SUBAPPLICATION GetEndpointFromOrchestrationOpcUaFull (* Get the endpoint at INDEX from a request orchestration response *)
  (* Standard: 61499-2; Description: Copyright (c) 2019 fortiss GmbH This program and the accompanying materials are made available under the terms of the Eclipse Public License 2.0 which is available at https://www.eclipse.org/legal/epl-2.0/ SPDX-License-Identifier: EPL-2.0 *)
  (* Version 1.0, 2019-09-17, Jose Cabral, fortiss GmbH *)
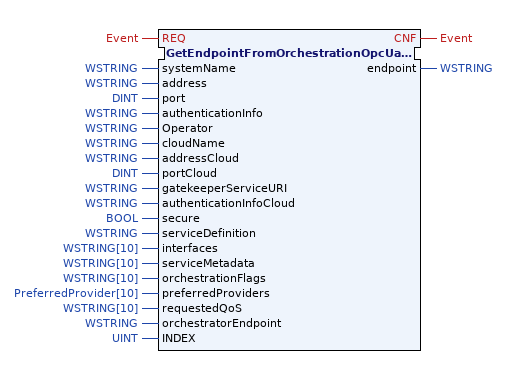
  EVENT_INPUT
    REQ; (* Request orchestration *)
  END_EVENT
  EVENT_OUTPUT
    CNF; (* Request finished *)
  END_EVENT
  VAR_INPUT
    systemName : WSTRING; (* Identification of the system *)
    address : WSTRING; (* Address of the offered services *)
    port : DINT; (* Port of the of the offered services *)
    authenticationInfo : WSTRING; (* Authentication info of the system *)
    Operator : WSTRING; (* Company (the capital  O is to avoid clash when exporting to C++) *)
    cloudName : WSTRING; (* Identification of the cloud *)
    addressCloud : WSTRING; (* Address to access the cloud *)
    portCloud : DINT; (* Port to access the cloud *)
    gatekeeperServiceURI : WSTRING; (* (Unclear documentation) *)
    authenticationInfoCloud : WSTRING; (* Authentication info of the cloud *)
    secure : BOOL; (* (Unclear documentation) *)
    serviceDefinition : WSTRING; (* Identification of the service *)
    interfaces : ARRAY [0..9] OF WSTRING; (* Interfaces implemented by the service *)
    serviceMetadata : ARRAY [0..9] OF WSTRING; (* Metadata of the service in key=value format *)
    orchestrationFlags : ARRAY [0..9] OF WSTRING; (* These flags can be set to tailor the orchestration process (use just the names of the flags to be enabled) *)
    preferredProviders : ARRAY [0..9] OF PreferredProvider; (* There can be a list from the Consumer stating which other Application Systems (even from other Clouds) it wishes to connect. If this field is filled out, the Orchestrator will try to facilitate these preferences *)
    requestedQoS : ARRAY [0..9] OF WSTRING; (* This object will be presenting the Consumer’s selected QoS level. Not implemented *)
    orchestratorEndpoint : WSTRING; (* Enpoint of the orchestrator *)
    INDEX : UINT; (* Position in the array of the requested forms *)
  END_VAR
  VAR_OUTPUT
    endpoint : WSTRING; (* Endpoint at position INDEX from orchestration forms *)
  END_VAR
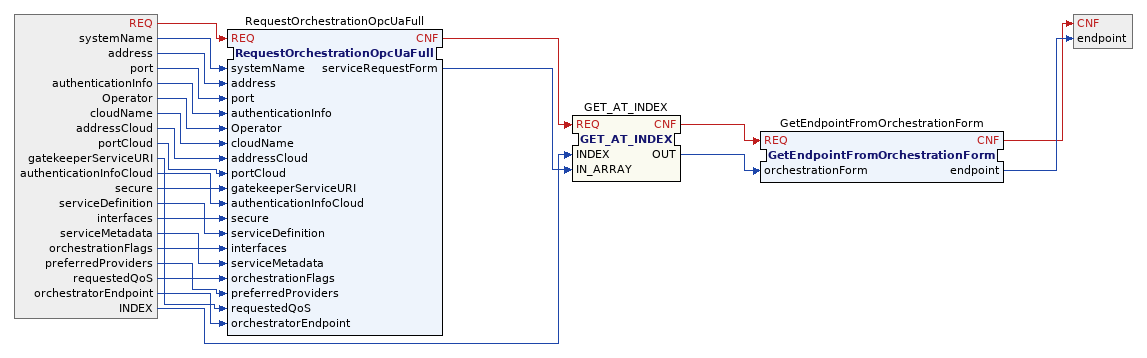
  FBS
    GET_AT_INDEX : GET_AT_INDEX;
  END_FBS
  SUBAPPS
    GetEndpointFromOrchestrationForm : GetEndpointFromOrchestrationForm;
    RequestOrchestrationOpcUaFull : RequestOrchestrationOpcUaFull;
  END_SUBAPPS
  EVENT_CONNECTIONS
    GET_AT_INDEX.CNF TO GetEndpointFromOrchestrationForm.REQ;
    GetEndpointFromOrchestrationForm.CNF TO CNF;
    REQ TO RequestOrchestrationOpcUaFull.REQ;
    RequestOrchestrationOpcUaFull.CNF TO GET_AT_INDEX.REQ;
  END_CONNECTIONS
  DATA_CONNECTIONS
    GET_AT_INDEX.OUT TO GetEndpointFromOrchestrationForm.orchestrationForm;
    INDEX TO GET_AT_INDEX.INDEX;
    GetEndpointFromOrchestrationForm.endpoint TO endpoint;
    systemName TO RequestOrchestrationOpcUaFull.systemName;
    address TO RequestOrchestrationOpcUaFull.address;
    port TO RequestOrchestrationOpcUaFull.port;
    authenticationInfo TO RequestOrchestrationOpcUaFull.authenticationInfo;
    Operator TO RequestOrchestrationOpcUaFull.Operator;
    cloudName TO RequestOrchestrationOpcUaFull.cloudName;
    addressCloud TO RequestOrchestrationOpcUaFull.addressCloud;
    portCloud TO RequestOrchestrationOpcUaFull.portCloud;
    gatekeeperServiceURI TO RequestOrchestrationOpcUaFull.gatekeeperServiceURI;
    authenticationInfoCloud TO RequestOrchestrationOpcUaFull.authenticationInfoCloud;
    secure TO RequestOrchestrationOpcUaFull.secure;
    serviceDefinition TO RequestOrchestrationOpcUaFull.serviceDefinition;
    interfaces TO RequestOrchestrationOpcUaFull.interfaces;
    serviceMetadata TO RequestOrchestrationOpcUaFull.serviceMetadata;
    orchestrationFlags TO RequestOrchestrationOpcUaFull.orchestrationFlags;
    preferredProviders TO RequestOrchestrationOpcUaFull.preferredProviders;
    requestedQoS TO RequestOrchestrationOpcUaFull.requestedQoS;
    orchestratorEndpoint TO RequestOrchestrationOpcUaFull.orchestratorEndpoint;
    RequestOrchestrationOpcUaFull.serviceRequestForm TO GET_AT_INDEX.IN_ARRAY;
  END_CONNECTIONS
END_SUBAPPLICATION
